# EPICS substitutions: viocs/si_ps/si_psApp/Db/sd1j.substitutions
file "db/individual.db" {
    pattern { family, pos }
        { "SD1J", "01C1" }
        { "SD1J", "02C1" }
        { "SD1J", "03C1" }
        { "SD1J", "04C1" }
        { "SD1J", "05C1" }
        { "SD1J", "06C1" }
        { "SD1J", "07C1" }
        { "SD1J", "08C1" }
        { "SD1J", "09C1" }
        { "SD1J", "10C1" }
        { "SD1J", "11C1" }
        { "SD1J", "12C1" }
        { "SD1J", "13C1" }
        { "SD1J", "14C1" }
        { "SD1J", "15C1" }
        { "SD1J", "16C1" }
        { "SD1J", "17C1" }
        { "SD1J", "18C1" }
        { "SD1J", "19C1" }
        { "SD1J", "20C1" }
}
